// TIA Portal V16 export
// export: Created 2021-07-12T14:47:21.0406743Z, ExportSetting WithDefaults, DisplayName Totally Integrated Automation Portal, DisplayVersion V16, DisplayName TIA Portal Version Control Interface, DisplayVersion V16, DisplayName TIA Portal Openness, DisplayVersion V16, DisplayName STEP 7 Professional, DisplayVersion V16, DisplayName STEP 7 Safety, DisplayVersion V16, DisplayName WinCC Professional, DisplayVersion V16
TYPE "SimaHydTO_typeHMIConnectionVCharSelectorCommand"
TITLE = SimaHydTO_typeHMIConnectionVCharSelectorCommand
// HMI interface: Hydraulic characteristics (VChar) selection of VChar array - Command (HMI -> PLC)
// stored: IsFailsafeCompliant false
   STRUCT
      previousObject : Bool;
      nextObject : Bool;
      executeDirectIndexSelection : Bool;
      directIndexSelection : Int;
   END_STRUCT;
END_TYPE
